{attribute 'GeneratedUsingTerminal: EL2911-0000-0016'}
{attribute addProperty BoxType "EL2911-0000-0016"}
{attribute addProperty Id "Module_1_FSOEModule_1_FSOE_7E34DB4019Module_2_FSOUTModule_2_FSOUT_1E8D16371Module_3_DEVICEIOModule_3_DEVICEIO_5FA6B4E72Module_4_FSLOGICModule_4_FSLOGIC_DEAB45222WcStateAT %I*WcState_B516A2644InfoDataAT %I*InfoData_94A18F5E2"}
{attribute addProperty CRC "3605533250"}
{attribute addProperty Size "30"}
TYPE EL2911_D6E81242 EXTENDS EtcSlaveTerminalBase_947E5A46 :
STRUCT
	{attribute addProperty Name "Module_1_FSOE"}
	Module_1_FSOE : Module_1_FSOE_7E34DB40;
	{attribute addProperty Name "Module_2_FSOUT"}
	Module_2_FSOUT : Module_2_FSOUT_1E8D1637;
	{attribute addProperty Name "Module_3_DEVICEIO"}
	Module_3_DEVICEIO : Module_3_DEVICEIO_5FA6B4E7;
	{attribute addProperty Name "Module_4_FSLOGIC"}
	Module_4_FSLOGIC : Module_4_FSLOGIC_DEAB4522;
	{attribute addProperty Name "WcState"}
	WcState : WcState_B516A264;
	{attribute addProperty Name "InfoData"}
	InfoData : InfoData_94A18F5E;
END_STRUCT
END_TYPE

(* stored: Version 1.2.0.0, ProductVersion 3.1.4024.9
   DUT EL2911_D6E81242: Id {0452db12-970b-4ade-8891-0dfcfb553034} *)
